Fanuc KAREL source: kx00005.KL

-- PROVISIONAL review KL for V770-1; original PC SHA256 3642639989a36a982e8360f3bad1d49dcfdf0b0b86d69f105114406a697dcb93
-- Incomplete behavior may be omitted. Consult companion uncertainty JSON. Do not deploy.
PROGRAM KX00005
%NOLOCKGROUP
VAR
  I : INTEGER
  J : INTEGER
  B : BOOLEAN
  F : FILE
  S : STRING[80]
-- UNRESOLVED_DECL P type=000102
BEGIN
  -- UNRESOLVED_PC offsets 5-32; opcodes 22,3F,3F,3D
  -- UNRESOLVED_PC offsets 37-44; opcodes 22,A3
  -- UNRESOLVED_PC offsets 49-56; opcodes 22,39
  -- UNRESOLVED_PC offsets 61-65; opcodes 7F
END KX00005
